// Mitsubishi GX Works2 project: example_fx   PLC: FX3U/FX3UC

PROGRAM MAIN
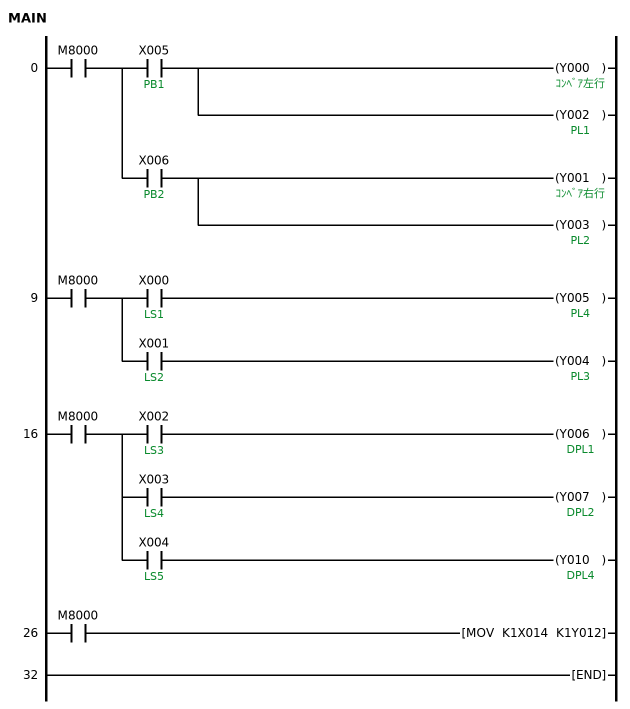
0     LD      M8000
      MPS
      AND     X005  ; PB1
      OUT     Y000  ; ｺﾝﾍﾞｱ左行
      OUT     Y002  ; PL1
      MPP
      AND     X006  ; PB2
      OUT     Y001  ; ｺﾝﾍﾞｱ右行
      OUT     Y003  ; PL2
9     LD      M8000
      MPS
      AND     X000  ; LS1
      OUT     Y005  ; PL4
      MPP
      AND     X001  ; LS2
      OUT     Y004  ; PL3
16    LD      M8000
      MPS
      AND     X002  ; LS3
      OUT     Y006  ; DPL1
      MRD
      AND     X003  ; LS4
      OUT     Y007  ; DPL2
      MPP
      AND     X004  ; LS5
      OUT     Y010  ; DPL4
26    LD      M8000
      MOV     K1X014 K1Y012  ; DSW1 / DPL10
32    END
END_PROGRAM

// device comments not shown above
X007  ; PB3
X010  ; PB4
X011  ; PB5
X013  ; 自動/手動
X015  ; DSW2
X016  ; DSW4
X017  ; DSW8
M100  ; ｺﾝﾍﾞｱ左行
M101  ; PL1
M102  ; ｺﾝﾍﾞｱ右行
M103  ; PL2
M200  ; PL3
M201  ; ｺﾝﾍﾞｱ左行
M202  ; ｺﾝﾍﾞｱ右行
Y011  ; DPL8
Y013  ; DPL20
Y014  ; DPL40
Y015  ; DPL80
